FUNCTION_BLOCK FB_FieldCodecInt32 IMPLEMENTS I_FieldCodec
VAR_INPUT
END_VAR
VAR_OUTPUT
END_VAR
VAR
    nValue : UDINT;
END_VAR

METHOD IsPackedRepeatedField : BOOL
VAR_INPUT
	nTag	: UDINT;
END_VAR
IsPackedRepeatedField := F_IsPackedRepeatedField(nTag);
END_METHOD


METHOD ValueReader : HRESULT
VAR_IN_OUT CONSTANT
	aBuffer	: ARRAY [*] OF BYTE;
END_VAR
VAR_IN_OUT
	stState	: ST_ParserInternalState;
END_VAR
VAR_OUTPUT
	anyOut	: T_Any;
END_VAR

ValueReader := F_ParseRawVarint32(aBuffer, stState, nValue);
anyOut := F_ToAnyType(anyArg:= nValue);
END_METHOD

{warning 'Add method implementation '}
{attribute 'analysis' := '-33'}
METHOD ValueWriter : HRESULT
VAR_IN_OUT
	aBuffer	: ARRAY [*] OF BYTE;
END_VAR
VAR_IN_OUT
	stState	: ST_WriterInternalState;
END_VAR
VAR_INPUT
	anyIn	: ANY;
END_VAR
END_METHOD

END_FUNCTION_BLOCK

(* stored: Version 1.1.0.1
   POU FB_FieldCodecInt32: Id {8bd84137-9243-445a-82a1-5a30e5da42ae}, SpecialFunc None
   Method IsPackedRepeatedField: Id {99247b5c-9995-4689-95f2-8e7ca845c7ef}
   Method ValueReader: Id {f0e2f0a6-ad5d-4700-b47f-c0159be5e107}
   Method ValueWriter: Id {3b271a1e-cec2-4f7c-b69e-965369e26732} *)
